// TIA Portal V18 export
DATA_BLOCK "ST10Cylinder"   // DB1020
{ S7_Optimized_Access := 'FALSE' }
// stored: AutoNumber false
   VAR RETAIN
      Cy { S7_SetPoint := 'True'} : Array[1..110] of "Cyl";
   END_VAR
BEGIN
   // Cy[1] : A-顶升模组-01阻挡气缸
   // Cy[2] : A-顶升模组-01升降气缸
   // Cy[3] : A-顶升模组-02阻挡气缸
   // Cy[4] : A-顶升模组-02升降气缸
   // Cy[5] : A-托盘缓存阻挡气缸
   // Cy[6] : C-贴标模组水平移动Y轴
   // Cy[7] : C-贴标模组垂直移动Z轴
   // Cy[8] : C-贴标模组螺标签切料真空吸附
   // Cy[9] : C-贴标模组标签取料真空吸附-02
   // Cy[10] : C-贴标模组换型气缸
   Cy[1..10].In.Error := false;
   Cy[1..10].In.GoWorkInterlock := false;
   Cy[1..10].In.GoHomeInterlock := false;
   Cy[1..10].In.WorkPositionSensor := false;
   Cy[1..10].In.HomePositionSensor := false;
   Cy[1].In.ValveType := false;
   Cy[2].In.ValveType := true;
   Cy[3].In.ValveType := false;
   Cy[4].In.ValveType := true;
   Cy[5].In.ValveType := false;
   Cy[6..10].In.ValveType := true;
   Cy[1..10].In.ManualOutputType := false;
   Cy[1..10].In.FaultTime := 50;
   Cy[1..10].In.OnPositionTime := 10;
   Cy[1..10].Inout.ManualGoWork := FALSE;
   Cy[1..10].Inout.ManualGoHome := FALSE;
   Cy[1..10].Inout.AutoGoWork := FALSE;
   Cy[1..10].Inout.AutoGoHome := FALSE;
   Cy[1..10].S.GoWorkTime := 0;
   Cy[1..10].S.GoHomeTime := 0;
   Cy[1..10].S.WorkFaultTime := 0;
   Cy[1..10].S.HomeFaultTime := 0;
   Cy[1..10].S.BothSensorOnTime := 0;
   Cy[1..10].S.Pulse100mSP := FALSE;
   Cy[1..10].S.AutoGoWorkP := FALSE;
   Cy[1..10].S.AutoGoHomeP := FALSE;
   Cy[1..10].S.GoWork100mSP := TRUE;
   Cy[1..10].S.GoHome100mSP := TRUE;
   Cy[1..10].S.BothSensorOn100mSP := TRUE;
   Cy[1..10].S.Alarm := FALSE;
   Cy[1..10].S.spare1 := FALSE;
   Cy[1..10].S.spare2 := 16#00;
   Cy[1..10].Out.GoWorkPosition := FALSE;
   Cy[1].Out.GoHomePosition := FALSE;
   Cy[2].Out.GoHomePosition := TRUE;
   Cy[3].Out.GoHomePosition := FALSE;
   Cy[4].Out.GoHomePosition := TRUE;
   Cy[5..10].Out.GoHomePosition := FALSE;
   Cy[1..9].Out.GoWPButtonActive := TRUE;
   Cy[10].Out.GoWPButtonActive := FALSE;
   Cy[1..9].Out.GoHPButtonActive := TRUE;
   Cy[10].Out.GoHPButtonActive := FALSE;
   Cy[1..10].Out.GoWorkFault := FALSE;
   Cy[1..10].Out.GoHomeFault := FALSE;
   Cy[1..10].Out.SensorPositionFault := FALSE;
   Cy[1].Out.CyNO := 16#01;
   Cy[2].Out.CyNO := 16#02;
   Cy[3].Out.CyNO := 16#03;
   Cy[4].Out.CyNO := 16#04;
   Cy[5].Out.CyNO := 16#05;
   Cy[6].Out.CyNO := 16#06;
   Cy[7].Out.CyNO := 16#07;
   Cy[8].Out.CyNO := 16#08;
   Cy[9].Out.CyNO := 16#09;
   Cy[10].Out.CyNO := 16#0A;
END_DATA_BLOCK
